FUNCTION_BLOCK FB_NanotecPD_Home
VAR_INPUT
	bExecute 	: BOOL;
	bStop		: BOOL;
END_VAR
VAR_OUTPUT
	bBusy 		: BOOL;
	bError 		: BOOL;
	nErrorId 	: ERRORID;	
END_VAR
VAR_IN_OUT
	pHwRef : POINTER TO FB_HwRefNanotecPD; 
END_VAR
VAR
	nState 				: USINT;
	nStateNext			: USINT;
	fbSdoWrite 			: FB_SDO_WRITE;
	eCurrentHomingState : E_CoDS402HomingState;
END_VAR

IF bExecute THEN
	CASE nState OF
		0:	//Set fast homing speed
			bBusy := TRUE;
			fbSdoWrite.nIndex := 16#6099;
			fbSdoWrite.nSubIndex := 1;
			fbSdoWrite.nDataLength := 4;
			fbSdoWrite.nData := pHwRef^.M_RealToInternSpeed(pHwRef^.P_nFastHomingSpeed);
			nState := 40;
			nStateNext := 1;
			
		1:	//Set slow homing speed
			fbSdoWrite.nIndex := 16#6099;
			fbSdoWrite.nSubIndex := 2;
			fbSdoWrite.nDataLength := 4;
			fbSdoWrite.nData := pHwRef^.M_RealToInternSpeed(pHwRef^.P_nSlowHomingSpeed);
			nState := 40;
			nStateNext := 2;
			
		2:	//Set homing methode
			fbSdoWrite.nIndex := 16#6098;
			fbSdoWrite.nSubIndex := 0;
			fbSdoWrite.nDataLength := 1;
			IF pHwRef^.P_bInvertInitDir THEN
				fbSdoWrite.nData := 2;
			ELSE
				fbSdoWrite.nData := 1;
			END_IF
			nState := 40;
			nStateNext := 3;
			
		3: 	//Write home offset
			fbSdoWrite.nIndex := 16#607C;
			fbSdoWrite.nSubIndex := 0;
			fbSdoWrite.nDataLength := 4;
			//Hier braucht es Umrechnung von Real to intern Pos
			fbSdoWrite.nData := pHwRef^.M_RealToInternPos(pHwRef^.P_nRefPos);
			nState := 40;
			IF pHwRef^.M_GetDS402State() = E_CoDS402States.DS402STATE_OperationEnabled THEN
				nStateNext := 4;
			ELSE
				nStateNext := 5;
			END_IF
			
		4:	//Mode lässt sich nicht in "OperationEnabled" setzen
			pHwRef^.nControlword := 7;
			IF pHwRef^.M_GetDS402State() = E_CoDS402States.DS402STATE_SwitchedOn THEN
				nState := 5;	
			END_IF
			
		5:	//Set Mode of operation to "6" (Homing)
			pHwRef^.nMode := 6; //Homing
			IF pHwRef^.nCurrentMode = 6 THEN
				nState := 6;	
			END_IF

		6:	//Statemachine in "OperationEnabled" setzen
			pHwRef^.nControlword := 15;
			IF pHwRef^.M_GetDS402State() = E_CoDS402States.DS402STATE_OperationEnabled THEN
				nState := 7;
			END_IF
			
		7:	//Start homing
			pHwRef^.nControlword := 31;
			eCurrentHomingState := pHwRef^.M_GetHomingState();
			IF eCurrentHomingState = E_CoDS402HomingState.HomingInProgress THEN
				nState := 8;
			END_IF
			
		8:	//Wait for State "Homing in process
			IF pHwRef^.M_GetDS402State() = E_CoDS402States.DS402STATE_OperationEnabled THEN
				IF bStop THEN
					pHwRef^.nControlword := 15;
					nState := 80;
				ELSE
					eCurrentHomingState := pHwRef^.M_GetHomingState();
					CASE eCurrentHomingState OF
						E_CoDS402HomingState.HomingAttainedButNotReached,
						E_CoDS402HomingState.HomingError,
						E_CoDS402HomingState.HomingInteruptedOrNotReached:
							nErrorId := E_ErrorIdDS402.ERRORID_HomingInterruptedOrNotReached;
							nState := 99;
						E_CoDS402HomingState.HomingSuccess:
							pHwRef^.P_bIsHomed := TRUE;
							pHwRef^.nControlword := 7;
							pHwRef^.nMode := 1;
							pHwRef^.nTargetSpeed := DINT_TO_INT(pHwRef^.M_RealToInternSpeed(pHwRef^.P_nFastHomingSpeed));
							pHwRef^.nTargetPosition := pHwRef^.M_RealToInternPos(pHwRef^.P_nHomePos);
							nState := 9;
					END_CASE
				END_IF
			ELSE
				nErrorId := E_ErrorIdDS402.ERRORID_OperationNotEnabled;
				nState := 99;
			END_IF
			
		9:	//Move to WorkingPos1
			IF pHwRef^.nCurrentMode = 1 THEN
				pHwRef^.nControlword := 15;
				nState := 10;
			END_IF
			
		10:	IF pHwRef^.M_GetDS402State() = E_CoDS402States.DS402STATE_OperationEnabled THEN
				pHwRef^.nControlword := 31;
				nState := 11;
			END_IF
			
		11:	//Wait for setpoint acknowledge
			IF pHwRef^.nStatusword.12 THEN
				pHwRef^.nControlword := 15;
				nState := 12;
			END_IF
			
		12:	//Wait for target reached
			IF pHwRef^.M_GetDS402State() = E_CoDS402States.DS402STATE_OperationEnabled THEN
				IF bStop THEN
					pHwRef^.nControlword.8 := TRUE;
					nState := 13;
				ELSE
					IF pHwRef^.nStatusword.10 THEN
						nState := 80;	
					END_IF
				END_IF
			ELSE
				nErrorId := E_ErrorIdDS402.ERRORID_OperationNotEnabled;
				nState := 99;
			END_IF
			
		13:	//Warten bis Motor sich nicht mehr dreht -> dann Power-STM in SwitchedOn setzen, damit Fahrauftrag gelöscht wird
			IF pHwRef^.nCurrentSpeed = 0 THEN
				pHwRef^.nControlword := 7;
				nState := 14;
			END_IF
			
		14:	//Power-STM wieder in OperationEnable setzen
			IF pHwRef^.M_GetDS402State() = E_CoDS402States.DS402STATE_SwitchedOn THEN
				pHwRef^.nControlword := 15;
				pHwRef^.P_bIsHomed := TRUE;
				nState := 80;
			END_IF		

	END_CASE
	
	//Sdo senden
	IF nState = 40 THEN
		fbSdoWrite(sADSNetID:= pHwRef^.P_sAdsNetId, nPortNr:= pHwRef^.P_nAdsPort, bExecute:= TRUE);
		IF NOT fbSdoWrite.bBusy THEN
			IF fbSdoWrite.bError THEN
				nErrorId := fbSdoWrite.nAdsErrorId;
				nState := 99;
			ELSE
				nState := nStateNext;
			END_IF
			fbSdoWrite(bExecute:= FALSE);
		END_IF		
	END_IF
	
	IF nState >= 80 THEN
		bBusy := FALSE;
		IF nState = 99 THEN
			bError := TRUE;
		END_IF
	END_IF
	
ELSE
	bError := FALSE;
	nErrorId := 0;
	nState := 0;	
END_IF

END_FUNCTION_BLOCK

(* stored: Version 1.1.0.1, ProductVersion 3.1.4024.11
   POU FB_NanotecPD_Home: Id {e62114fb-8409-4c13-8c17-7a6a8283316b}, SpecialFunc None *)
